// TwinCAT 3 PLC project KL6781_MBus
// ProgramVersion: 3.1.4024.12
// libraries:
//   Tc2_MBus, * (Beckhoff Automation GmbH)
//   Tc2_Standard, * (Beckhoff Automation GmbH)
//   Tc2_System, * (Beckhoff Automation GmbH)
//   Tc3_Module, * (Beckhoff Automation GmbH)
// project tree:
//   GVLs/ GVL_IO.TcGVL
//   / PlcTask.TcTTO, PlcTask_Fast.TcTTO
//   POUs/ MAIN.TcPOU, P_MBus.TcPOU, P_MBus_Fast.TcPOU

CONFIGURATION KL6781_MBus
    RESOURCE PLC ON TwinCAT3
        TASK PlcTask(INTERVAL := T#10ms, PRIORITY := 30);
        TASK PlcTask_Fast(INTERVAL := T#2ms, PRIORITY := 9);
        PROGRAM MAIN WITH PlcTask : MAIN;
        PROGRAM P_MBus_Fast WITH PlcTask_Fast : P_MBus_Fast;
    END_RESOURCE
END_CONFIGURATION

// ---- GVLs/GVL_IO.TcGVL
{attribute 'qualified_only'}
VAR_GLOBAL
    stComIn    AT %I* : ST_KL6781inData22B;
    stComOut   AT %Q* : ST_KL6781outData22B;
    stCom             : ST_MBUS_Communication;
END_VAR

// ---- POUs/MAIN.TcPOU
PROGRAM MAIN
VAR
END_VAR

P_MBus();

END_PROGRAM

// ---- POUs/P_MBus.TcPOU
PROGRAM P_MBus
VAR
	fbMBUS_EMU_32x7		: FB_MBUS_EMU_32x7;
END_VAR

fbMBUS_EMU_32x7(
	usiAddress			:= 15, 					// MBus address of the meter
	stSecAdr			:= , 					// Only used if you address via the secundairy address
	eBaudrate			:= , 					// Default setting = 2400
	bStart				:= , 					// A raising edge will trigger a single read
	bSND_NKE			:= , 					
	bReadInit			:= , 					// Trigger a read when the PLC starts
	tMinSendTime		:= , 					// Default = 2s --> update time for automatic reading
	usiUnit				:= , 					// Unit of the energy values to be output by the block. 0=W(h) / 1=KW(h) / 2 =MW(h) / 3=GW(h)
	bDisabled			:= , 
	bBusy				=> , 
	bReady				=> , 
	bError				=> , 
	eError				=> , 
	dwIdNumber			=> , 
	byStatus			=> , 
	byGEN				=> , 
	byCounter			=> , 
	usiRecivedAdr		=> , 
	eMedium				=> , 
	sMan				=> , 
	stOperatingHours	=> , 					// Data from meter
	stEnergy			=> ,  					// Data from meter
	stPower				=> ,  					// Data from meter
	stInitCounter		=> ,  					// Data from meter
	stDeviceError		=> , 
	stCom				:= GVL_IO.stCom);

END_PROGRAM

// ---- POUs/P_MBus_Fast.TcPOU
PROGRAM P_MBus_Fast
VAR
	fbMBUSKL6781		: FB_MBUSKL6781;
END_VAR

fbMBUSKL6781(
	usiRetries	:= , 
	bStart		:= , 
	bDisabled	:= , 
	bBusy		=> , 
	bReady		=> , 
	bError		=> , 
	eError		=> , 
	stComIn		:= GVL_IO.stComIn, 
	stComOut	:= GVL_IO.stComOut, 
	stCom		:= GVL_IO.stCom);

END_PROGRAM
